{attribute 'qualified_only'}
VAR_GLOBAL CONSTANT INTERNAL
    cTagTypeBits : UINT := 3;
    cTagTypeMask : UINT := 7;   // (1 << cTagTypeBits) - 1;
END_VAR

(* stored: Version 1.1.0.1
   GVL GCL_WireFormat: Id {ed0e2fb5-2b5e-40b9-abc2-01f63cd9771f} *)
